// Mitsubishi GX Works2 project: ServMotor2   PLC: Q03UDV

PROGRAM MAIN
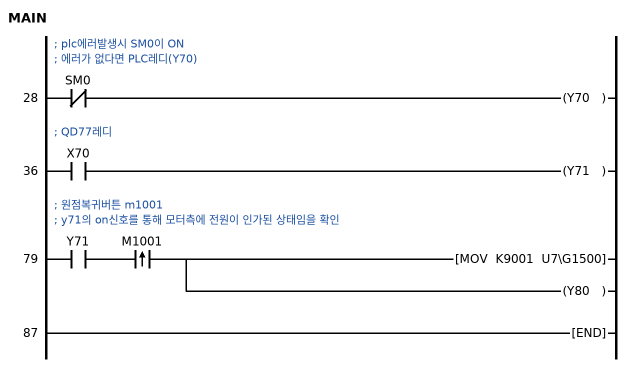
; plc에러발생시 SM0이 ON
; 에러가 없다면 PLC레디(Y70)
28    LDI     SM0
      OUT     Y70
; QD77레디
36    LD      X70
      OUT     Y71
; 원점복귀버튼 m1001
; y71의 on신호를 통해 모터측에 전원이 인가된 상태임을 확인
79    LD      Y71
      ANDP    M1001
      MOV     K9001 U7\G1500
      OUT     Y80
87    END
END_PROGRAM
